DATA_BLOCK "bioVal.D"
TITLE = Batch I/O Value Data Block
{ S7_Optimized_Access := 'TRUE' }
AUTHOR : Woermann
VERSION : 1.0
// -- Woermann Automation --
// Date: 2020-06-20
NON_RETAIN
   VAR RETAIN
      Val : Array[0..15] of "bioVal.DT";
   END_VAR

BEGIN

END_DATA_BLOCK

